(* PLC project KinIn_v3.project, CODESYS CODESYS V3.5 SP19 *)
(* stored: creationDateTime 2025-01-20T16:27:00.2066936, modificationDateTime 2025-01-20T16:17:39.6822999 *)

FUNCTION_BLOCK Eye
  VAR_INPUT
    {attribute 'variable_length_array_original_scope' := 'Inout'}
    {attribute 'variable_length_array' := 'ARRAY[*,*] OF REAL'}
    {attribute 'Dimensions' := '2'}
    eye : POINTER TO REAL;
  END_VAR
  VAR
    i : DINT;
    j : DINT;
  END_VAR

            FOR i:=1 TO UPPER_BOUND(eye,1) DO
	FOR j:=1 TO UPPER_BOUND(eye,1) DO
		IF i=j THEN
			eye[i,j]:=1;
		ELSE		
			eye[i,j]:=0;
		END_IF
	END_FOR
END_FOR
          
END_FUNCTION_BLOCK
